PROGRAM MAIN
VAR
	bJustASimpleBoolean : BOOL; // SA0033 - WARNING
	sThisStringIsTooLong : STRING(6) := 'Hello world'; // SA0026 - ERROR
	
	nCounter : ULINT;
END_VAR

nCounter := nCounter + 1;

sThisStringIsTooLong := '';

END_PROGRAM

(* stored: Version 1.1.0.1, ProductVersion 3.1.4022.12
   POU MAIN: Id {45fa1b65-8964-4d83-bf67-fe76a4f119d2}, SpecialFunc None *)
